TYPE ST_WaferTransferRequest :
STRUCT
	Send : ST_WaferTransferCtrl;
	Receive : ST_WaferTransferCtrl;
END_STRUCT
END_TYPE

(* stored: Version 1.1.0.1, ProductVersion 3.1.4026.18
   DUT ST_WaferTransferRequest: Id {c286521e-06fc-4b3c-8036-193bb81c9317} *)
